{attribute 'GeneratedUsingTerminal: EL3773-0000-0016'}
{attribute addProperty BoxType "EL3773-0000-0016"}
{attribute addProperty Id "StartTimeNextLatchAT %I*ULINT8"}
{attribute addProperty CRC "2600321653"}
{attribute addProperty Size "8"}
TYPE AI_Timestamp_NextSync1Time_9AFDC275 :
STRUCT
	{attribute addProperty Name "StartTimeNextLatch"}
	StartTimeNextLatch AT %I* : ULINT;
END_STRUCT
END_TYPE

(* stored: Version 1.2.0.0, ProductVersion 3.1.4024.9
   DUT AI_Timestamp_NextSync1Time_9AFDC275: Id {9889d3a9-2c57-4f2d-bc37-cd179c671f54} *)
